// TIA Portal project "palatizer 17.07" (V15)
// Vorlageprojekt für das Buch mit Zielsystem S7-1200

(* hardware
DEVICE "S7-1200-Station_1"  S7-1200 Station
   slot 0: "Baugruppenträger_0"  Rack  V1.0
   slot 1: "PLC_1"  CPU 1211C DC/DC/DC  6ES7 211-1AE40-0XB0  V4.1
DEVICE "S7-1200 station_1"  S7-1200 Station
   slot 0: "Rack_0"  S7-1200 Rack  Rack  V1.0
   slot 1: "PLC_2"  CPU 1214C DC/DC/DC  6ES7 214-1AG40-0XB0  V4.2
*)

// ===== PLC "PLC_1"  CPU 1211C DC/DC/DC =====

VAR_GLOBAL   // PLC tag table "Standard-Variablentabelle"
   "pallet feeder" AT %Q0.0 : Bool;
   "load pallet" AT %Q0.1 : Bool;
   "exit conveyor" AT %Q0.2 : Bool;
   "move to limit" AT %Q0.3 : Bool;
   "elevator up" AT %Q0.4 : Bool;
   "elevator down" AT %Q0.5 : Bool;
   "box feeder" AT %Q0.6 : Bool;
   "turn" AT %Q0.7 : Bool;
   "push" AT %Q1.0 : Bool;
   "load belt" AT %Q1.1 : Bool;
   "clamp" AT %Q1.2 : Bool;
   "open plate" AT %Q1.3 : Bool;
   "warning light" AT %Q1.4 : Bool;
   "start light" AT %Q1.5 : Bool;
   "reset light" AT %Q1.6 : Bool;
   "stop light" AT %Q1.7 : Bool;
   "pallet at entry" AT %I0.0 : Bool;
   "pallet at exit" AT %I0.1 : Bool;
   "pallet loaded" AT %I0.2 : Bool;
   "box at entry" AT %I0.3 : Bool;
   "pusher limit" AT %I0.4 : Bool;
   "plate limit" AT %I0.5 : Bool;
   "clamped" AT %I0.6 : Bool;
   "elevator moving" AT %I0.7 : Bool;
   "start" AT %I1.0 : Bool;
   "reset" AT %I1.1 : Bool;
   "stop" AT %I1.2 : Bool;
   "emergency stop" AT %I1.3 : Bool;
   "auto" AT %I1.4 : Bool;
   "RUN" AT %I1.5 : Bool;
   "Tag_1" AT %M0.5 : Bool;
   "Tag_2" AT %M0.2 : Bool;
   "Tag_3" AT %M2.0 : Bool;
   "Tag_4" AT %M3.0 : Bool;
END_VAR

// folder: System blocks/Program resources

DATA_BLOCK "push tp"   // DB1
{ S7_Optimized_Access := 'TRUE' }
AUTHOR : Simatic
FAMILY : IEC
NAME : IEC_TMR
VERSION : 1.0
// stored: InstanceOfName IEC_TIMER
"IEC_TIMER"
BEGIN
END_DATA_BLOCK

DATA_BLOCK "palet bekleme"   // DB2
{ S7_Optimized_Access := 'TRUE' }
AUTHOR : Simatic
FAMILY : IEC
NAME : IEC_TMR
VERSION : 1.0
// stored: InstanceOfName IEC_TIMER
"IEC_TIMER"
BEGIN
END_DATA_BLOCK

DATA_BLOCK "IEC_Timer_0_DB"   // DB3
{ S7_Optimized_Access := 'TRUE' }
AUTHOR : Simatic
FAMILY : IEC
NAME : IEC_TMR
VERSION : 1.0
// stored: InstanceOfName IEC_TIMER
"IEC_TIMER"
BEGIN
END_DATA_BLOCK

DATA_BLOCK "box counter"   // DB4
{ S7_Optimized_Access := 'TRUE' }
AUTHOR : Simatic
FAMILY : IEC
NAME : CNTR
VERSION : 1.0
// stored: InstanceOfName IEC_COUNTER
"IEC_COUNTER"
BEGIN
END_DATA_BLOCK

DATA_BLOCK "IEC_Timer_0_DB_1"   // DB5
{ S7_Optimized_Access := 'TRUE' }
AUTHOR : Simatic
FAMILY : IEC
NAME : IEC_TMR
VERSION : 1.0
// stored: InstanceOfName IEC_TIMER
"IEC_TIMER"
BEGIN
END_DATA_BLOCK

DATA_BLOCK "palet durdurma"   // DB6
{ S7_Optimized_Access := 'TRUE' }
AUTHOR : Simatic
FAMILY : IEC
NAME : IEC_TMR
VERSION : 1.0
// stored: InstanceOfName IEC_TIMER
"IEC_TIMER"
BEGIN
END_DATA_BLOCK

DATA_BLOCK "kutu yukleme tp"   // DB7
{ S7_Optimized_Access := 'TRUE' }
AUTHOR : Simatic
FAMILY : IEC
NAME : CNTR
VERSION : 1.0
// stored: InstanceOfName IEC_COUNTER
"IEC_COUNTER"
BEGIN
END_DATA_BLOCK

DATA_BLOCK "kutu yukleme geciktirme"   // DB8
{ S7_Optimized_Access := 'TRUE' }
AUTHOR : Simatic
FAMILY : IEC
NAME : IEC_TMR
VERSION : 1.0
// stored: InstanceOfName IEC_TIMER
"IEC_TIMER"
BEGIN
END_DATA_BLOCK

DATA_BLOCK "open palet"   // DB9
{ S7_Optimized_Access := 'TRUE' }
AUTHOR : Simatic
FAMILY : IEC
NAME : IEC_TMR
VERSION : 1.0
// stored: InstanceOfName IEC_TIMER
"IEC_TIMER"
BEGIN
END_DATA_BLOCK

DATA_BLOCK "clamp bkleme"   // DB10
{ S7_Optimized_Access := 'TRUE' }
AUTHOR : Simatic
FAMILY : IEC
NAME : IEC_TMR
VERSION : 1.0
// stored: InstanceOfName IEC_TIMER
"IEC_TIMER"
BEGIN
END_DATA_BLOCK

DATA_BLOCK "indirme bekletmesi"   // DB11
{ S7_Optimized_Access := 'TRUE' }
AUTHOR : Simatic
FAMILY : IEC
NAME : IEC_TMR
VERSION : 1.0
// stored: InstanceOfName IEC_TIMER
"IEC_TIMER"
BEGIN
END_DATA_BLOCK

DATA_BLOCK "kapak kapatma bekletici"   // DB12
{ S7_Optimized_Access := 'TRUE' }
AUTHOR : Simatic
FAMILY : IEC
NAME : IEC_TMR
VERSION : 1.0
// stored: InstanceOfName IEC_TIMER
"IEC_TIMER"
BEGIN
END_DATA_BLOCK

DATA_BLOCK "kapak acma sayici"   // DB13
{ S7_Optimized_Access := 'TRUE' }
AUTHOR : Simatic
FAMILY : IEC
NAME : CNTR
VERSION : 1.0
// stored: InstanceOfName IEC_COUNTER
"IEC_COUNTER"
BEGIN
END_DATA_BLOCK

DATA_BLOCK "palet indirme gecikme"   // DB14
{ S7_Optimized_Access := 'TRUE' }
AUTHOR : Simatic
FAMILY : IEC
NAME : IEC_TMR
VERSION : 1.0
// stored: InstanceOfName IEC_TIMER
"IEC_TIMER"
BEGIN
END_DATA_BLOCK

DATA_BLOCK "palet cikis"   // DB15
{ S7_Optimized_Access := 'TRUE' }
AUTHOR : Simatic
FAMILY : IEC
NAME : IEC_TMR
VERSION : 1.0
// stored: InstanceOfName IEC_TIMER
"IEC_TIMER"
BEGIN
END_DATA_BLOCK

DATA_BLOCK "dongu"   // DB16
{ S7_Optimized_Access := 'TRUE' }
AUTHOR : Simatic
FAMILY : IEC
NAME : IEC_TMR
VERSION : 1.0
// stored: InstanceOfName IEC_TIMER
"IEC_TIMER"
BEGIN
END_DATA_BLOCK

DATA_BLOCK "palet dongu"   // DB17
{ S7_Optimized_Access := 'TRUE' }
AUTHOR : Simatic
FAMILY : IEC
NAME : IEC_TMR
VERSION : 1.0
// stored: InstanceOfName IEC_TIMER
"IEC_TIMER"
BEGIN
END_DATA_BLOCK

DATA_BLOCK "palet 2 durdurma"   // DB18
{ S7_Optimized_Access := 'TRUE' }
AUTHOR : Simatic
FAMILY : IEC
NAME : IEC_TMR
VERSION : 1.0
// stored: InstanceOfName IEC_TIMER
"IEC_TIMER"
BEGIN
END_DATA_BLOCK

DATA_BLOCK "asansör beklme"   // DB19
{ S7_Optimized_Access := 'TRUE' }
AUTHOR : Simatic
FAMILY : IEC
NAME : IEC_TMR
VERSION : 1.0
// stored: InstanceOfName IEC_TIMER
"IEC_TIMER"
BEGIN
END_DATA_BLOCK

DATA_BLOCK "palet sayıcı"   // DB20
{ S7_Optimized_Access := 'TRUE' }
AUTHOR : Simatic
FAMILY : IEC
NAME : CNTR
VERSION : 1.0
// stored: InstanceOfName IEC_COUNTER
"IEC_COUNTER"
BEGIN
END_DATA_BLOCK

DATA_BLOCK "load pallet kesme"   // DB21
{ S7_Optimized_Access := 'TRUE' }
AUTHOR : Simatic
FAMILY : IEC
NAME : IEC_TMR
VERSION : 1.0
// stored: InstanceOfName IEC_TIMER
"IEC_TIMER"
BEGIN
END_DATA_BLOCK

DATA_BLOCK "c2"   // DB22
{ S7_Optimized_Access := 'TRUE' }
AUTHOR : Simatic
FAMILY : IEC
NAME : CNTR
VERSION : 1.0
// stored: InstanceOfName IEC_COUNTER
"IEC_COUNTER"
BEGIN
END_DATA_BLOCK

DATA_BLOCK "load pallet kesme2"   // DB23
{ S7_Optimized_Access := 'TRUE' }
AUTHOR : Simatic
FAMILY : IEC
NAME : IEC_TMR
VERSION : 1.0
// stored: InstanceOfName IEC_TIMER
"IEC_TIMER"
BEGIN
END_DATA_BLOCK

DATA_BLOCK "IEC_Counter_0_DB"   // DB24
{ S7_Optimized_Access := 'TRUE' }
AUTHOR : Simatic
FAMILY : IEC
NAME : CNTR
VERSION : 1.0
// stored: InstanceOfName IEC_COUNTER
"IEC_COUNTER"
BEGIN
END_DATA_BLOCK

DATA_BLOCK "1snlik gecikme"   // DB25
{ S7_Optimized_Access := 'TRUE' }
AUTHOR : Simatic
FAMILY : IEC
NAME : IEC_TMR
VERSION : 1.0
// stored: InstanceOfName IEC_TIMER
"IEC_TIMER"
BEGIN
END_DATA_BLOCK

// folder: (top level)

FUNCTION "MHJ-PLC-Lab-Function-S71200" : Void   // FC9000, SCL
{ S7_Optimized_Access := 'TRUE' }
VERSION : 0.1
   VAR_TEMP
      rdTimeReturn : Int;
      outputTime : DTL;
      SyncVal : Byte;
      forVal : Int;
      forVal_2 : Int;
      Value : Byte;
   END_VAR
   VAR CONSTANT
      CompVal : Byte := 16#34;
      Value_01 : Byte := 16#11;
      Value_01_DW : DWord := 16#A165_D992;
      Value_02_DW : DWord := 16#58BE_4401;
   END_VAR
BEGIN

   #Value:=PEEK(area := 16#82,
        dbNumber := 0,
        byteOffset := 511);
   #Value := #Value + 1;

   POKE(area := 16#82,
        dbNumber := 0,
        byteOffset := 511,
        value := #Value);

   POKE(area:=16#81,
        dbNumber:=0,
        byteOffset:=1016,
        value:=#Value_01_DW);
   POKE(area := 16#81,
        dbNumber := 0,
        byteOffset := 1020,
        value := #Value_02_DW);

   POKE(area := 16#81,
        dbNumber := 0,
        byteOffset := 511,
        value := B#16#00);

   FOR #forVal := 0 TO 120 DO
       FOR #forVal_2:=0 TO 10 DO
           #rdTimeReturn:=RD_SYS_T(#outputTime);
           #rdTimeReturn := WR_SYS_T(#outputTime);
           #rdTimeReturn := RD_SYS_T(#outputTime);
           #rdTimeReturn := WR_SYS_T(#outputTime);
       END_FOR;
       #SyncVal:= PEEK(area := 16#81,
                      dbNumber := 0,
                      byteOffset := 511);
       IF #SyncVal = #CompVal THEN
          GOTO M_1;
       END_IF;
   END_FOR;
   RETURN;

   M_1:
   POKE(area := 16#81,
        dbNumber := 0,
        byteOffset := 511,
        value := B#16#0);
END_FUNCTION

ORGANIZATION_BLOCK "Main"   // OB1, LAD, ProgramCycle
TITLE = "Main Program Sweep (Cycle)"
{ S7_Optimized_Access := 'TRUE' }
VERSION : 0.1
   VAR_INPUT
      Initial_Call : Bool;   // Initial call of this OB
      Remanence : Bool;   // =True, if remanent data are available
   END_VAR
   VAR_TEMP   // added for the SCL form of the ladder/FBD networks
      _w1 : Bool;
   END_VAR
BEGIN

REGION Network 1
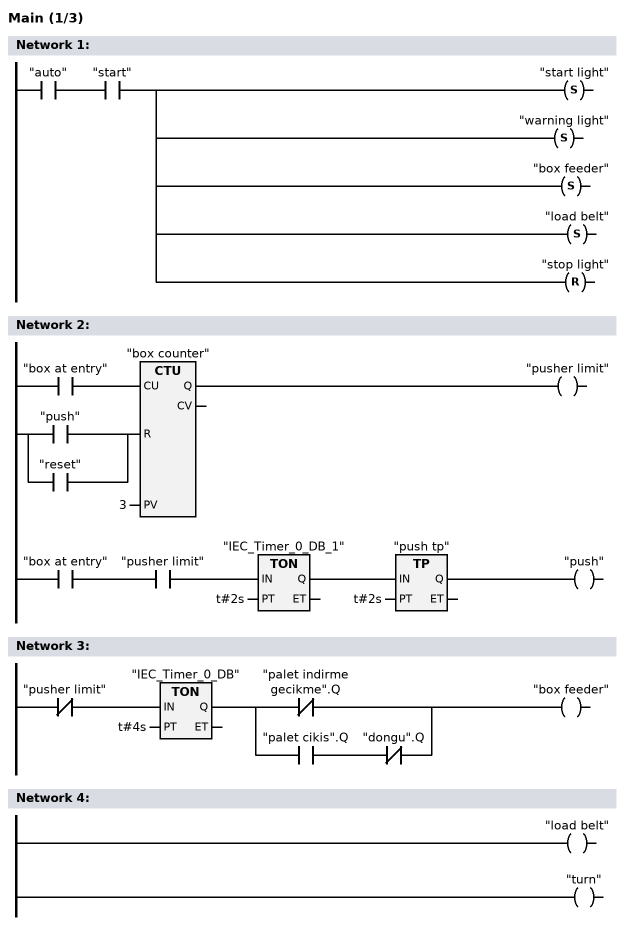
   RUNG wire#powerrail
      Contact( "auto" )
      Contact( "start" )
      wire#w1
      S_Coil( "start light" )
   END_RUNG
   RUNG wire#w1
      S_Coil( "warning light" )
   END_RUNG
   RUNG wire#w1
      S_Coil( "box feeder" )
   END_RUNG
   RUNG wire#w1
      S_Coil( "load belt" )
   END_RUNG
   RUNG wire#w1
      R_Coil( "stop light" )
   END_RUNG
   // the same network as SCL:
   IF "auto" AND "start" THEN
       "start light" := TRUE;
       "warning light" := TRUE;
       "box feeder" := TRUE;
       "load belt" := TRUE;
       "stop light" := FALSE;
   END_IF;
END_REGION

REGION Network 2
   "box counter".CTU(CU := "box at entry", R := "push" OR "reset", PV := 3);
   "pusher limit" := "box counter".Q;
   "IEC_Timer_0_DB_1".TON(IN := "box at entry" AND "pusher limit", PT := t#2s);
   "push tp".TP(IN := "IEC_Timer_0_DB_1".Q, PT := t#2s);
   "push" := "push tp".Q;
END_REGION

REGION Network 3
   "IEC_Timer_0_DB".TON(IN := NOT "pusher limit", PT := t#4s);
   "box feeder" := "IEC_Timer_0_DB".Q AND (NOT "palet indirme gecikme".Q OR ("palet cikis".Q AND NOT "dongu".Q));
END_REGION

REGION Network 4
   RUNG wire#powerrail
      Coil( "load belt" )
   END_RUNG
   RUNG wire#powerrail
      Coil( "turn" )
   END_RUNG
   // the same network as SCL:
   "load belt" := TRUE;
   "turn" := TRUE;
END_REGION

REGION Network 6
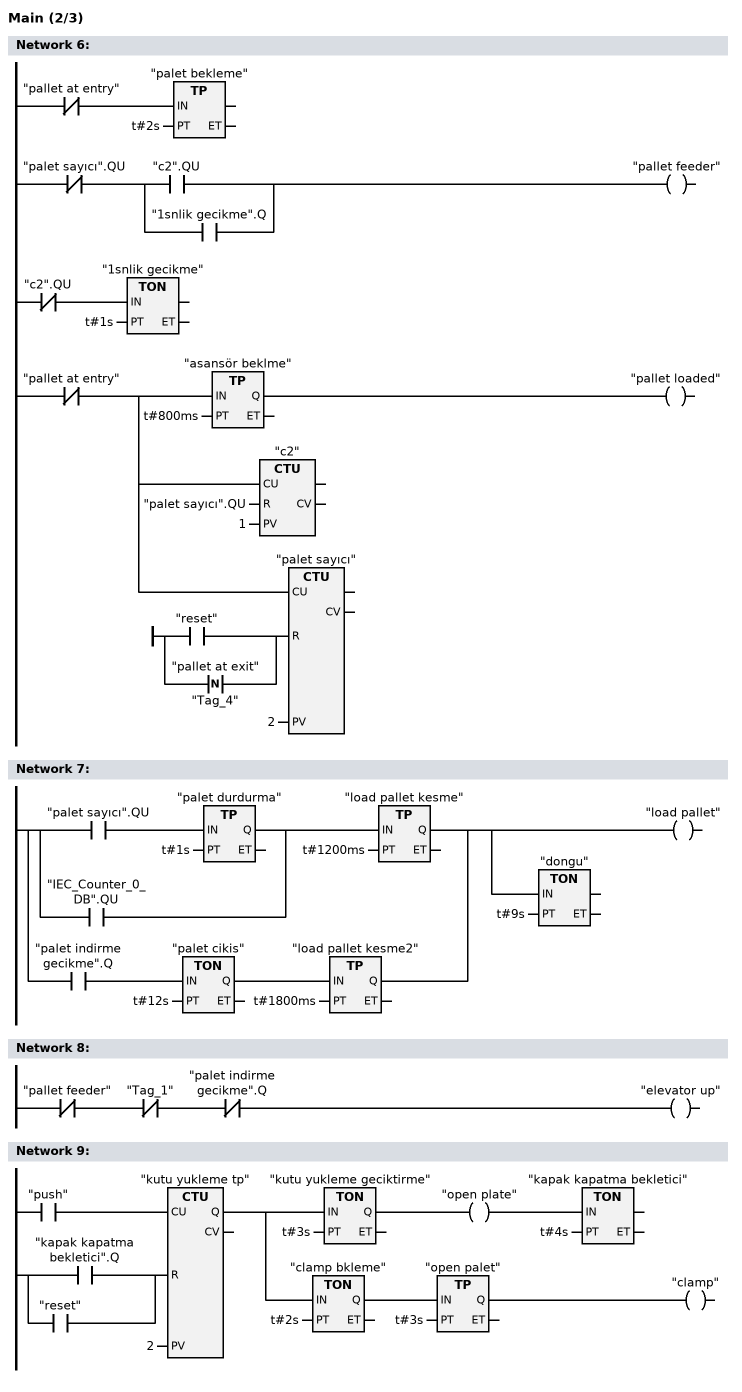
   "palet bekleme".TP(IN := NOT "pallet at entry", PT := t#2s);
   "pallet feeder" := NOT "palet sayıcı".QU AND ("c2".QU OR "1snlik gecikme".Q);
   "1snlik gecikme".TON(IN := NOT "c2".QU, PT := t#1s);
   "asansör beklme".TP(IN := NOT "pallet at entry", PT := t#800ms);
   "pallet loaded" := "asansör beklme".Q;
   "c2".CTU(CU := NOT "pallet at entry", R := "palet sayıcı".QU, PV := 1);
   #_w1 := NOT "pallet at exit" AND "Tag_4";   // falling edge of "pallet at exit"
   "Tag_4" := "pallet at exit";
   "palet sayıcı".CTU(CU := NOT "pallet at entry", R := "reset" OR #_w1, PV := 2);
END_REGION

REGION Network 7
   "palet durdurma".TP(IN := "palet sayıcı".QU, PT := t#1s);
   "load pallet kesme".TP(IN := "palet durdurma".Q OR "IEC_Counter_0_DB".QU, PT := t#1200ms);
   "palet cikis".TON(IN := "palet indirme gecikme".Q, PT := t#12s);
   "load pallet kesme2".TP(IN := "palet cikis".Q, PT := t#1800ms);
   "load pallet" := "load pallet kesme".Q OR "load pallet kesme2".Q;
   "dongu".TON(IN := "load pallet", PT := t#9s);
END_REGION

REGION Network 8
   RUNG wire#powerrail
      I_Contact( "pallet feeder" )
      I_Contact( "Tag_1" )
      I_Contact( "palet indirme gecikme".Q )
      Coil( "elevator up" )
   END_RUNG
   // the same network as SCL:
   "elevator up" := NOT "pallet feeder" AND NOT "Tag_1" AND NOT "palet indirme gecikme".Q;
END_REGION

REGION Network 9
   "kutu yukleme tp".CTU(CU := "push", R := "kapak kapatma bekletici".Q OR "reset", PV := 2);
   "kutu yukleme geciktirme".TON(IN := "kutu yukleme tp".Q, PT := t#3s);
   "open plate" := "kutu yukleme geciktirme".Q;
   "kapak kapatma bekletici".TON(IN := "kutu yukleme geciktirme".Q, PT := t#4s);
   "clamp bkleme".TON(IN := "kutu yukleme tp".Q, PT := t#2s);
   "open palet".TP(IN := "clamp bkleme".Q, PT := t#3s);
   "clamp" := "open palet".Q;
END_REGION

REGION Network 10
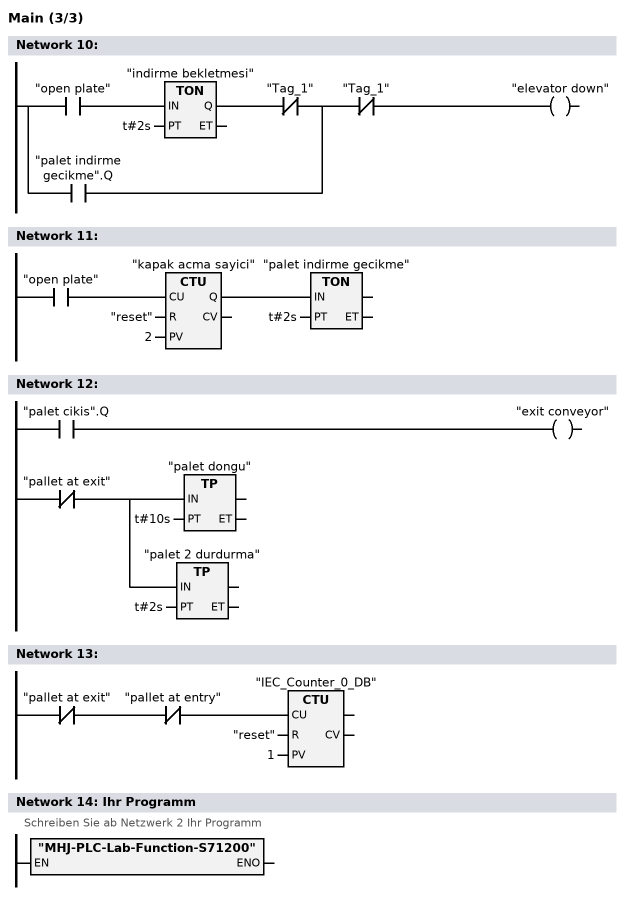
   "indirme bekletmesi".TON(IN := "open plate", PT := t#2s);
   "elevator down" := (("indirme bekletmesi".Q AND NOT "Tag_1") OR "palet indirme gecikme".Q) AND NOT "Tag_1";
END_REGION

REGION Network 11
   "kapak acma sayici".CTU(CU := "open plate", R := "reset", PV := 2);
   "palet indirme gecikme".TON(IN := "kapak acma sayici".Q, PT := t#2s);
END_REGION

REGION Network 12
   "exit conveyor" := "palet cikis".Q;
   "palet dongu".TP(IN := NOT "pallet at exit", PT := t#10s);
   "palet 2 durdurma".TP(IN := NOT "pallet at exit", PT := t#2s);
END_REGION

REGION Network 13
   "IEC_Counter_0_DB".CTU(CU := NOT "pallet at exit" AND NOT "pallet at entry", R := "reset", PV := 1);
END_REGION

REGION Network 14: Ihr Programm
   // Schreiben Sie ab Netzwerk 2 Ihr Programm
   RUNG wire#powerrail
      "MHJ-PLC-Lab-Function-S71200"()
   END_RUNG
   // the same network as SCL:
   "MHJ-PLC-Lab-Function-S71200"();
END_REGION
END_ORGANIZATION_BLOCK

// ===== PLC "PLC_2"  CPU 1214C DC/DC/DC =====

ORGANIZATION_BLOCK "Main"   // OB1, LAD, ProgramCycle
TITLE = "Main Program Sweep (Cycle)"
{ S7_Optimized_Access := 'TRUE' }
VERSION : 0.1
   VAR_INPUT
      Initial_Call : Bool;   // Initial call of this OB
      Remanence : Bool;   // =True, if remanent data are available
   END_VAR
BEGIN
END_ORGANIZATION_BLOCK